(* PLC project KinIn_v3.project, CODESYS CODESYS V3.5 SP19 *)
(* stored: creationDateTime 2025-01-20T16:23:09.9752867, modificationDateTime 2025-01-20T16:17:39.6822999 *)

FUNCTION_BLOCK angVelToSkewSymMatrix
  VAR_INPUT
    omg : ARRAY[1..3] OF REAL;  (* 3vector *)
  END_VAR
  VAR_OUTPUT
    so3mat : ARRAY[1..3, 1..3] OF REAL;  (* 3x3matrix *)
  END_VAR

            //fast is just plain assignment
so3mat[1,1]:=0;
so3mat[1,2]:=-omg[3];
so3mat[1,3]:=omg[2];
so3mat[2,1]:=omg[3];
so3mat[2,2]:=0;
so3mat[2,3]:=-omg[1];
so3mat[3,1]:=-omg[2];
so3mat[3,2]:=omg[1];
so3mat[3,3]:=0;
          
END_FUNCTION_BLOCK
